(* CoDeSys 2.3.9.59 project: Esercizio 1.pro *)
(* Libraries: STANDARD.LIB *)

(* Task configuration *)
TASK Standard (PRIORITY := 0, INTERVAL := T#10ms);
	ESERCIZIO
END_TASK

(* POU ESERCIZIO, LD *)
PROGRAM ESERCIZIO
VAR
	Presenza_Pezzo AT %IX0.0: BOOL;
	Pistone_Indietro AT %IX0.4: BOOL;
	Pistone_Avanti AT %IX0.2: BOOL;
	Fine_Corsa AT %IX0.6: BOOL;

	Nastro_On AT %QX0.0: BOOL;
	Pistone_On AT %QX0.2: BOOL;

	Movimento_Giostra AT %QX3.4: BOOL;
	Trapano_Down AT %QX7.0: BOOL;

	Timer_Pistone: TON;
	Timer_Nastro: TON;
	Stop_Nastro: BOOL;
	Pezzo_Giostra: BOOL;
	Giostra_BUSY AT %IX6.1: BOOL;

END_VAR
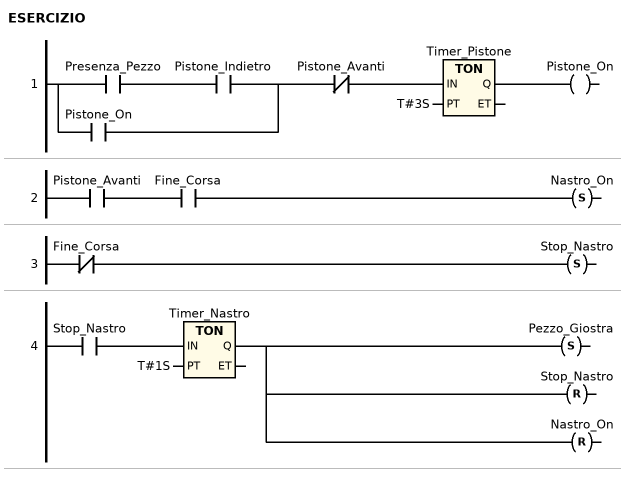
_LD_ (* Ladder Diagram *)
NETWORK 1
	{ [Presenza_Pezzo] - [Pistone_Indietro] | [Pistone_On] } - [/Pistone_Avanti] - Timer_Pistone:TON(IN: *, PT: T#3S) --- (Pistone_On)
NETWORK 2
	[Pistone_Avanti] - [Fine_Corsa] --- (S Nastro_On)
NETWORK 3
	[/Fine_Corsa] --- (S Stop_Nastro)
NETWORK 4
	[Stop_Nastro] - Timer_Nastro:TON(IN: *, PT: T#1S) --- (S Pezzo_Giostra) (R Stop_Nastro) (R Nastro_On)
_END_LD_
(* the same logic as Structured Text *)
(* Network 1 *)
Timer_Pistone(IN := (Presenza_Pezzo AND Pistone_Indietro OR Pistone_On) AND NOT Pistone_Avanti, PT := T#3S);
Pistone_On := Timer_Pistone.Q;
(* Network 2 *)
IF Pistone_Avanti AND Fine_Corsa THEN Nastro_On := TRUE; END_IF;
(* Network 3 *)
IF NOT Fine_Corsa THEN Stop_Nastro := TRUE; END_IF;
(* Network 4 *)
Timer_Nastro(IN := Stop_Nastro, PT := T#1S);
IF Timer_Nastro.Q THEN Pezzo_Giostra := TRUE; Stop_Nastro := FALSE; Nastro_On := FALSE; END_IF;
END_PROGRAM
